{attribute 'qualified_only'}
VAR_GLOBAL
END_VAR

(* stored: Version 1.1.0.1, ProductVersion 3.1.4022.7
   GVL GVL_01_Station: Id {6318a88d-7aaa-4558-87ef-0982c3f79d5b} *)
